Yaskawa INFORM job: R2_W28-29-A1(180,180)_MP_OK.JBI

/JOB
//NAME R2_W28-29-A1(180,180)_MP_OK
///FOLDERNAME MP_TEST
//POS
///NPOS 57,57,0,3,0,0
///TOOL 0
///POSTYPE PULSE
///PULSE
C00000=80119,-26538,-45313,94350,88003,22329
C00001=25991,22819,-44384,62089,90781,34609
C00002=38364,-75513,-108384,55989,71493,-7325
C00003=35055,-151610,-110006,56580,73793,-34788
C00004=81331,-134370,-85628,49597,55830,-34464
C00005=88203,-128135,-82461,48057,53099,-32115
C00006=93050,-123166,-83526,41761,55455,-27840
C00007=93973,-122952,-82755,41729,54749,-27694
C00008=90716,-125546,-81139,47335,52165,-31198
C00009=82685,-120655,-76340,53903,58521,-34985
C00010=83556,-119016,-75904,53568,58382,-34538
C00011=82685,-120655,-76340,53903,58521,-34985
C00012=79888,-122654,-77423,54209,59874,-35773
C00013=72406,-127274,-79988,54640,63607,-37743
C00014=70873,-107960,-82014,51148,71410,-33723
C00015=71222,-108949,-82435,51181,71056,52537
C00016=78020,-147139,-86256,61734,36188,84086
C00017=86485,-141156,-82447,58811,31667,87005
C00018=89614,-138661,-80886,57271,30071,88275
C00019=90628,-136843,-80546,55809,29919,89176
C00020=89614,-138661,-80886,57271,30071,88275
C00021=50763,-108918,-51550,78969,67439,76512
C00022=52905,-111216,-53010,79154,65432,76529
C00023=50763,-108918,-51550,78969,67439,76512
C00024=82293,-138770,-81921,56356,37936,87306
C00025=90309,-136226,-81433,52831,34135,90466
C00026=90310,-135115,-80106,53122,33983,90309
C00027=90309,-136226,-81433,52831,34135,90466
C00028=85948,-145790,-85360,57167,35051,87439
C00029=55072,-160435,-85881,65078,49179,76331
C00030=49607,-161929,-87270,64202,52302,75457
C00031=36202,-164957,-90678,61516,60027,73482
C00032=61211,-138193,-69550,92184,44447,32782
C00033=67762,-131025,-65030,93619,40218,33353
C00034=67908,-128348,-63402,93229,40118,33612
C00035=70055,-129679,-65001,93647,38715,33807
C00036=67765,-129497,-63219,94016,40226,33120
C00037=75326,-131354,-64124,97677,35398,32594
C00038=68087,-130814,-64994,93639,40005,33410
C00039=61606,-137994,-69521,92242,44191,32837
C00040=55258,-118108,-59725,86533,60293,52424
C00041=53813,-109348,-62526,74118,64386,70530
C00042=55148,-118183,-59739,86518,60364,52404
C00043=56049,-116883,-60583,86088,59882,53061
C00044=50641,-103746,-58230,73578,66553,70296
C00045=69135,-132595,-74868,74328,33950,54921
C00046=71098,-162548,-92117,95488,43349,66788
C00047=73820,-158062,-89714,95633,41530,67274
C00048=84872,-160122,-89024,105609,31341,66176
C00049=74755,-157498,-89648,93851,40243,69589
C00050=73722,-154029,-89200,91717,40906,70652
C00051=83420,-158789,-88106,104558,32228,66456
C00052=68934,-107867,-43642,78353,39539,88888
C00053=58723,-144124,-88388,37391,57840,66604
C00054=58723,-144124,-88388,37391,57840,66604
C00055=65119,-140602,-125961,30647,76298,75337
C00056=65119,-140602,-125961,59810,40226,75337
BC00000=326419,100109,1075213
BC00001=148486,153585,1075167
BC00002=155162,103003,1075170
BC00003=163791,37623,1075173
BC00004=169464,-5360,1075175
BC00005=169464,-5360,1075175
BC00006=169464,-5360,1075175
BC00007=169464,-5360,1075175
BC00008=169464,-5360,1075175
BC00009=169464,-5360,1075175
BC00010=169464,-5360,1075175
BC00011=169464,-5360,1075175
BC00012=169464,-5360,1075175
BC00013=169464,-5360,1075175
BC00014=180341,30737,1075175
BC00015=180341,30737,1075175
BC00016=188279,-5360,1075175
BC00017=188279,-5360,1075175
BC00018=188279,-5360,1075175
BC00019=188279,-5360,1075175
BC00020=188279,-5360,1075175
BC00021=188279,-5360,1075175
BC00022=188279,-5360,1075175
BC00023=188279,-5360,1075175
BC00024=188279,-5360,1075175
BC00025=188279,-5360,1075175
BC00026=188279,-5360,1075175
BC00027=188279,-5360,1075175
BC00028=188279,-5360,1075175
BC00029=188279,-36082,1075175
BC00030=188279,-36082,1075175
BC00031=188279,-36082,1075175
BC00032=166034,-5360,1075175
BC00033=165366,-5360,1075175
BC00034=165099,-5360,1075172
BC00035=165099,-5360,1075175
BC00036=165099,-5360,1075175
BC00037=135954,-5360,1075175
BC00038=131443,-5360,1075175
BC00039=132110,-5360,1075175
BC00040=140523,-5360,1071573
BC00041=134093,-5360,1075175
BC00042=138970,-5360,1066099
BC00043=138970,-5360,1066099
BC00044=134093,-5360,1075175
BC00045=120208,-5360,1075175
BC00046=191136,-5360,922686
BC00047=191136,-5360,922686
BC00048=189183,-5360,926090
BC00049=189183,-5360,926090
BC00050=189183,-5360,926090
BC00051=189183,-5360,926090
BC00052=174136,-5360,1074960
BC00053=177898,-5360,1043479
BC00054=177898,-5360,1043479
BC00055=165042,43182,1043479
BC00056=165042,304327,1043479
///POSTYPE BASE
///RECTAN
///RCONF 0,0,0,0,0,0,0,0,0,0,0,0,0,0,0,0,0,0,0,0,0,0,0,0
P00006=0.222,-3.123,-1.508,0.0000,0.0000,0.0000
P00022=0.222,-3.123,-1.508,0.0000,0.0000,0.0000
P00023=0.143,-0.036,0.682,0.0000,0.0000,0.0000
//INST
///DATE 2023/11/16 10:54
///ATTR SC,RW
///GROUP1 RB1,BS1
NOP
'r2_W28-29-A1(180,180)
'Path S925
COMM MOVJ C00000 BC00000 VJ=100.00
SFTOF
MOVJ C00001 BC00001 VJ=20.00
MOVJ C00002 BC00002 VJ=20.00
MOVJ C00003 BC00003 VJ=20.00
MOVL C00004 BC00004 V=100.0
MOVL C00005 BC00005 V=100.0
MOVL C00006 BC00006 V=60.0
REFP 3 C00007 BC00007
CALL JOB:SEARCH-R1
SET P023 P006
SFTON P023
MOVL C00008 BC00008 V=60.0
MOVL C00009 BC00009 V=60.0
REFP 3 C00010 BC00010
CALL JOB:SEARCH-R1
SET P023 P006
SFTON P023
MOVL C00011 BC00011 V=60.0
MOVL C00012 BC00012 V=100.0
MOVL C00013 BC00013 V=100.0
'Path VIA926
SFTOF
MOVJ C00014 BC00014 VJ=20.00
'Path VIA927
SFTOF
MOVJ C00015 BC00015 VJ=20.00
'Path S928
SFTOF
MOVJ C00016 BC00016 VJ=20.00
MOVL C00017 BC00017 V=100.0
MOVL C00018 BC00018 V=60.0
REFP 3 C00019 BC00019
CALL JOB:SEARCH-R1
SET P022 P006
SFTON P022
MOVL C00020 BC00020 V=60.0
MOVL C00021 BC00021 V=60.0
REFP 3 C00022 BC00022
CALL JOB:SEARCH-R1
SET P022 P006
SFTON P022
MOVL C00023 BC00023 V=60.0
MOVL C00024 BC00024 V=100.0
MOVL C00025 BC00025 V=60.0
REFP 3 C00026 BC00026
CALL JOB:SEARCH-R1
SET P022 P006
SFTON P022
MOVL C00027 BC00027 V=60.0
MOVL C00028 BC00028 V=100.0
COMM MOVL C00029 BC00029 V=100.0
COMM MOVL C00030 BC00030 V=400.0
COMM MOVL C00031 BC00031 V=1000.0
'Path W929
SFTOF
SFTON P022
MOVJ C00032 BC00032 VJ=20.00
MOVL C00033 BC00033 V=100.0
MOVL C00034 BC00034 V=100.0 PL=0
REFP 1 C00035 BC00035
REFP 2 C00036 BC00036
MACRO1 MJ#(0) ARGF7
ARCON
MOVL C00037 BC00037 V=10.0
ARCOF
MOVL C00038 BC00038 V=100.0
MOVL C00039 BC00039 V=100.0
SFTOF
'Path W930
SFTOF
SFTON P023
MOVL C00040 BC00040 V=100.0
MOVL C00041 BC00041 V=100.0 PL=0
REFP 1 C00042 BC00042
REFP 2 C00043 BC00043
MACRO1 MJ#(0) ARGF7
ARCON
MOVL C00044 BC00044 V=10.0
ARCOF
MOVL C00045 BC00045 V=100.0
SFTOF
'Path W931
SFTOF
SFTON P022
MOVL C00046 BC00046 V=166.7
MOVL C00047 BC00047 V=100.0
MOVL C00048 BC00048 V=100.0 PL=0
REFP 1 C00049 BC00049
REFP 2 C00050 BC00050
MACRO1 MJ#(0) ARGF7
'RUBAJ_NIE BYLO SPRAWDZONE KOLIZJ
ARCON
MOVL C00051 BC00051 V=10.0
MOVL C00052 BC00052 V=10.0
ARCOF
MOVL C00053 BC00053 V=100.0
MOVL C00054 BC00054 V=166.7
SFTOF
MOVJ C00055 BC00055 VJ=20.00
MOVJ C00056 BC00056 VJ=20.00
END
